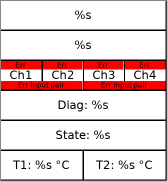
VISUALIZATION TplTsConnectionEL1904  // 168x182
VAR_IN_OUT
	stConnectionDiag 			:FB_TwinSafeConnectionEL1904;
END_VAR
(* End *)
    Rectangle (0,0 166x30), "%s", text variable: stConnectionDiag.sEcSlaveName, colour toggle: stConnectionDiag.sDiag = 'No error'
    Rectangle (0,60 42x30), "Ch1", colour toggle: stConnectionDiag.bChannel1
    Rectangle (42,60 42x30), "Ch2", colour toggle: stConnectionDiag.bChannel2
    Rectangle (83,60 42x30), "Ch3", colour toggle: stConnectionDiag.bChannel3
    Rectangle (124,60 42x30), "Ch4", colour toggle: stConnectionDiag.bChannel4
    Rectangle (0,90 166x30), "Diag: %s", text variable: stConnectionDiag.sDiag, colour toggle: stConnectionDiag.sDiag <> 'No error'
    Rectangle (0,120 166x30), "State: %s", text variable: stConnectionDiag.sState
    Rectangle (0,150 83x30), "T1: %s °C", text variable: stConnectionDiag.stSlaveTemp.nInternalTemperature1, colour toggle: stConnectionDiag.bTempWarning
    Rectangle (83,150 83x30), "T2: %s °C", text variable: stConnectionDiag.stSlaveTemp.nInternalTemperature2, colour toggle: stConnectionDiag.bTempWarning
    Rectangle (0,30 166x30), "%s", text variable: stConnectionDiag.sEcSlaveType
    Rectangle (84,81 81x8), "Err input pair", invisible if: NOT stConnectionDiag.stTsDiagObjectsBitsEL1904.bErrSecondInputPair
    Rectangle (1,61 40x8), "Err", invisible if: NOT stConnectionDiag.stTsDiagObjectsBitsEL1904.bErrInput1
    Rectangle (43,61 39x8), "Err", invisible if: NOT stConnectionDiag.stTsDiagObjectsBitsEL1904.bErrInput2
    Rectangle (84,61 39x8), "Err", invisible if: NOT stConnectionDiag.stTsDiagObjectsBitsEL1904.bErrInput3
    Rectangle (125,61 40x8), "Err", invisible if: NOT stConnectionDiag.stTsDiagObjectsBitsEL1904.bErrInput4
    Rectangle (1,81 81x8), "Err input pair", invisible if: NOT stConnectionDiag.stTsDiagObjectsBitsEL1904.bErrFirstInputPair
END_VISUALIZATION

(* stored: Version 1.1.0.1, ProductVersion 3.1.4024.11
   Visu TplTsConnectionEL1904: Id {09470d6c-fcc8-46ed-8b8c-331512b9619a} *)
